
// ===== library types =====

TYPE "LoadDataBlock"
VERSION : 0.1
   STRUCT
      data : Array[0..8192] of USInt;
   END_STRUCT;
END_TYPE

// ===== library: MasterCopy "ReadSDO" =====

FUNCTION_BLOCK "ReadSDO"   // FB104, SCL
{ S7_Optimized_Access := 'TRUE' }
VERSION : 0.1
   VAR_INPUT
      REQ : Bool;   // Start read SDO request
      ID : Word;   // Hardware ID of CM
      SLOT : Byte;   // Channel
      NODE : Int;   // Node ID
      INDEX : Word;   // Object index
      SUB : Byte;   // Object subindex
      DB : DInt;   // First memorybyte where recieved data is stored
   END_VAR
   VAR_OUTPUT
      SIZE : UInt;   // Size of recieved data
      BUSY : Bool;   // FB is busy
      RET : UInt;   // Result
   END_VAR
   VAR
      iState : Int;
      abResponseArray : Array[0..248] of Byte;
      abRequestArray : Array[0..4] of Byte;
      WriteSDO : WRREC;
      ReadSDO : RDREC;
      fReqWriteReadSDO : Bool;
      fReqReadSDO : Bool;
      fWriteReadSDOBusy : Bool;
      fReadSDOBusy : Bool;
      bSubindex : Byte;
      wReturn : Word;
      wErrorCode : Word;
      wNoHammeredSDO : Word;
      iDBIndex : Int;
      uiRequestTotalSize : UInt;
      iResponseDataSize : Int;
      uiResponseTotalSize : UInt;
      bAddErrInfo : Byte;
      dwStatus : DWord;
      fWriteReadSDOError : Bool;
      fWriteReadSDODone : Bool;
      fReadSDOValid : Bool;
      fReadSDOError : Bool;
      uiLen : UInt;
      wLen : Word;
      wTotLen : Word;
      fErrTooMuchSDOData : Bool;
      bNode : Byte;
      wIndex : Word;
      bSub : Byte;
      iReturnSize : Int;
      iDataIndex : Int;
      iResponseHeaderSize : Int;
      iReadLength : Int;
      iRecordNo : Int;
   END_VAR
   VAR_TEMP
      wTemp : Word;
      i : Int;
   END_VAR
BEGIN
   (* ------------------------------------------------------------------------
   Title:        Read SDO
   Description:  Block used for reading a single SDO from any CANopen node.
                 CM CANopen module needs to be in CANopen operation mode. 

   Author:       HMS
   Version:      1.0
   Date:         2013-05-29
      ------------------------------------------------------------------------ *)

   CASE #iState OF
     0:  // START
       IF #REQ THEN
         #BUSY                 :=  true;
         #fReqWriteReadSDO     :=  true;
         #fReqReadSDO          :=  true;

         #fErrTooMuchSDOData    :=  false;

         #fWriteReadSDOBusy    :=  false;
         #fReadSDOBusy         :=  false;

         #bNode                :=  INT_TO_BYTE(#NODE);
         #wIndex               :=  #INDEX;
         #bSub                 :=  #SUB;

         #abRequestArray[0]    :=  0;    //Frag byte
         #iReturnSize          :=  0;
         #iDataIndex           :=  0;

         #uiRequestTotalSize   :=  5;
         #iResponseHeaderSize  :=  9;
         #iResponseDataSize    :=  240;
         #uiResponseTotalSize  :=  249;
         #iRecordNo            :=  WORD_TO_INT(w#16#110);

         #iState               := 10;
     END_IF;

   10: //Check input parameter(s)
       IF #SLOT < 0 OR #SLOT > 7 THEN  // Index should be in the range 0 - 7
         #wReturn      :=  0;
         #bAddErrInfo  :=  B#16#4A;
         #iState       :=  900;  //Internal error
       ELSE
         #iRecordNo    :=  WORD_TO_INT(w#16#110+#SLOT);
         #iState       := 100;  //SDO
       END_IF;      

     100: //SDO
       #wNoHammeredSDO  :=  0;

       // Set up the Read SDO request
       #abRequestArray[1] :=  #bNode;
       #abRequestArray[2] :=  WORD_TO_BYTE(SHR(IN:=#wIndex,N:=8));
       #abRequestArray[3] :=  WORD_TO_BYTE(#wIndex);
       #abRequestArray[4] :=  #bSub;

      #iState   :=  110;

     110:  //Write
       #WriteSDO(
          REQ      :=  #fReqWriteReadSDO,
          ID       :=  #ID,
          INDEX    :=  #iRecordNo,
          LEN      :=  #uiRequestTotalSize,
          DONE     =>  #fWriteReadSDODone,
          BUSY     =>  #fWriteReadSDOBusy,
          ERROR    =>  #fWriteReadSDOError,
          STATUS   =>  #dwStatus,
          RECORD   :=  #abRequestArray
          );

       #fReqWriteReadSDO   :=  false;  // Reset variable to prevent this SFC from being called twice
       IF NOT #fWriteReadSDOBusy THEN
         #iState  := 120;
       END_IF;

     120:  //Evaluate writing
       #wReturn  :=  DWORD_TO_WORD(SHR(IN:=#dwStatus,N:=8)) AND W#16#FFFF;
       IF #fWriteReadSDOError THEN
         #iState  := 903;  //Write error
       ELSE  // Seems no error occured, continue with reading the SDO
         #iState  := 130;   //Read
       END_IF;

     130: //Read
      #ReadSDO(
       REQ       :=  #fReqReadSDO,
       ID        :=  #ID,
       INDEX     :=  #iRecordNo,
       MLEN      :=  #uiResponseTotalSize,
       VALID     =>  #fReadSDOValid,
       BUSY      =>  #fReadSDOBusy,
       ERROR     =>  #fReadSDOError,
       STATUS    =>  #dwStatus,
       LEN       =>  #uiLen,
       RECORD    :=  #abResponseArray
       );

       #fReqReadSDO :=  false;
       IF NOT #fReadSDOBusy THEN
         #iState  := 140;      
       END_IF;

     140:  //Evaluate reading, try again if failed
       #wTemp :=  DWORD_TO_WORD(SHR(IN:=#dwStatus,N:=8)) AND W#16#FFFF;
       IF #wTemp = W#16#80B5 OR #abResponseArray[0] =w#16#FE THEN
         #wNoHammeredSDO  :=  #wNoHammeredSDO + 1;
         IF #wNoHammeredSDO > 1000 THEN
          #wReturn  :=  0;
          #bAddErrInfo :=  b#16#13;
          #iState   := 900;  //Internal error
         ELSE
           #fReqReadSDO    :=  true;
           #iState         := 130;  //Read
         END_IF;
       ELSE
         #iState  := 150;  //CERR
       END_IF;

     150:  //CERR
       IF #fReadSDOError THEN  // Check for failure when sending the command
         #wReturn  :=  DWORD_TO_WORD(SHR(IN:=#dwStatus,N:=8)) AND W#16#FFFF;
         #iState      := 903;  //Read error
        ELSIF #abResponseArray[0] > 0 THEN // Check if the message was rejected by the module
         #wReturn  :=  B#16#FF;
         #bAddErrInfo  :=  #abResponseArray[0];
         #iState      := 903;  //Read error
       ELSE
         #iState  := 160;
     END_IF;

     160:  
       //
       #iReadLength :=  UINT_TO_INT(#uiLen) - #iResponseHeaderSize;
       #iReturnSize :=  #iReturnSize + #iReadLength;

       // Check for SDO error
       IF #abResponseArray[6] <> 0 THEN
         #bAddErrInfo  :=  #abResponseArray[6];
         #wReturn      :=  0;
         #iState       :=  903;
       ELSIF #iDataIndex >= #iResponseDataSize THEN    // Check if the data would be completely outside the array
         #iState       :=  300;  //CONT
       ELSIF (#iDataIndex + #iReadLength) <= #iResponseDataSize THEN
         #iState       :=  200;  //SOK
       ELSE
         #iReadLength  :=  #iResponseDataSize - #iDataIndex;
         #fErrTooMuchSDOData :=  true;
         #iState       :=  200;  //SOK
       END_IF;

     200:  //SOK
       // Copy data to the user-specified array
       FOR #i:=0 TO #iReadLength - 1 DO
         POKE(area       :=  16#84,
              dbNumber   :=  #DB,
              byteOffset :=  #iDataIndex + #i,
              value      :=  #abResponseArray[#iResponseHeaderSize + #i]);
       END_FOR;
       #iDataIndex   :=  #iDataIndex + #iReadLength;
       POKE(area       :=  16#84,
              dbNumber   :=  #DB,
              byteOffset :=  0,
              value      :=  #abResponseArray[#iResponseHeaderSize]);
       #iState       :=  300;  //CONT

     300:  //CONT
       //Check whether OR NOT TO CONTINUE

     // If this was the last message of a fragmented message, or this message was
     //  not fragmented at all, we're done
     IF (#abResponseArray[1] AND 1) = 0 OR (#abResponseArray[1] AND 2) > 0 THEN  
       #iState             := 400;  //DONE
     ELSE    // Not the last fragment, go again!
       #abRequestArray[1]  :=  #abResponseArray[1];
       #fReqWriteReadSDO   :=  true;
       #fReqReadSDO        :=  true;
       #iState             := 100;  //SDO
     END_IF;

     400:  //DONE
       IF #fErrTooMuchSDOData THEN
         #wErrorCode :=  W#16#22;
         #iState     :=  900;
       ELSE
         #RET    :=  0;
         #BUSY   :=  false;
         #SIZE   :=  INT_TO_UINT(#iReturnSize);
         #iState     :=  0;
       END_IF;

   (*** ERROR HANDLING ***)
     900:// Internal errors
       IF #wReturn = 0 AND #bAddErrInfo <> 0 THEN
         #wErrorCode :=  w#16#1000 + #bAddErrInfo;     
       ELSE
         #wErrorCode :=  W#16#FF00;  
       END_IF;
       #iState  := 999;

     903: //Range 3xxx (Read/Write errors)
       IF #wReturn = W#16#8090 THEN
         #wErrorCode :=  W#16#3100;
       ELSIF #wReturn = W#16#8093 THEN
         #wErrorCode :=  W#16#3200;
       ELSIF #wReturn = W#16#80A0 OR #wReturn = W#16#80A1 THEN
         #wErrorCode :=  W#16#3300;
       ELSIF #wReturn = W#16#80A2 THEN
         #wErrorCode :=  W#16#3701;
       ELSIF #wReturn = W#16#80A3 THEN
         #wErrorCode :=  W#16#3600;
       ELSIF #wReturn = W#16#80A4 THEN
         #wErrorCode :=  W#16#3702;
       ELSIF #wReturn = W#16#80B2 THEN
         #wErrorCode :=  W#16#3400;
       ELSIF #wReturn = W#16#80B3 THEN
         #wErrorCode :=  W#16#3500;
       ELSIF #wReturn >= W#16#80C1 AND #wReturn <= W#16#80C6 THEN
         #wErrorCode :=  #wReturn - W#16#80C0 + W#16#3702;
       ELSIF #wReturn = 0 THEN
         #wErrorCode :=  W#16#3800 + #bAddErrInfo;
       ELSIF #wReturn = W#16#FF THEN
         #wErrorCode :=  W#16#3900 + #bAddErrInfo;
       ELSE
         IF #wReturn <> 0 OR #bAddErrInfo = 0 THEN
           #wErrorCode :=  W#16#FF00;
         ELSE
           #wErrorCode :=  SHL(IN:=#bAddErrInfo, N:=8);
         END_IF;
       END_IF;
       #iState :=  999;

     999:
       IF #wErrorCode = 0 THEN
         #RET  :=  WORD_TO_UINT(w#16#FF00);
       ELSE
         #RET  :=  WORD_TO_UINT(#wErrorCode);
       END_IF;
       #SIZE   :=  INT_TO_UINT(#iReturnSize); 
       #BUSY   :=  false;
       #iState := 0;
   END_CASE;
END_FUNCTION_BLOCK

// ===== library: MasterCopy "CAN_CTRL" =====

FUNCTION_BLOCK "CAN_CTRL"   // FB1, SCL
{ S7_Optimized_Access := 'TRUE' }
VERSION : 0.1
   VAR_INPUT
      Req : Bool;
      ID : Word;
      FCN : Int;
      LEN : UInt;
      DB : DInt;
   END_VAR
   VAR_OUTPUT
      Busy : Bool;
      Ret : UInt;
   END_VAR
   VAR
      Read : RDREC;
      Write : WRREC;
      iState : Int;
      fReqWriteCmd : Bool;
      fWriteCmdDone : Bool;
      fWriteCmdBusy : Bool;
      fWriteCmdError : Bool;
      dwStatus : DWord;
      abRequest : Array[0..244] of Byte;
      fReqReadCmd : Bool;
      fReadCmdValid : Bool;
      fReadCmdBusy : Bool;
      fReadCmdError : Bool;
      uiLen : UInt;
      abResponse : Array[0..247] of Byte;
      iResonseHeaderSize : Int := 3;
      iResponseDataSize : Int := 245;
      uiResponseTotalSize : UInt := 248;
      wReturn : Word;
      bAddErrInfo : Byte;
      wNoHammered : Word;
      wErrorCode : Word;
      fHasMoreFragments : Bool;
      wParamLength : Word;
      uiCmdLength : UInt;
      wCOBIDsWritten : Word;
      bFragSegment : Byte;
      iOffset : Int;
      wLength : Word;
      iRecordNo : Int;
   END_VAR
   VAR_TEMP
      wTempStatus : Word;
      wTemp : Word;
      i : Int;
   END_VAR
BEGIN
   (* ------------------------------------------------------------------------
   Title:        CAN Control
   Description:  Block used for controlling a CM CANopen 
                 module in transparent mode

   Author:       HMS
   Version:      1.0
   Date:         2013-05-25
      ------------------------------------------------------------------------ *)

   CASE #iState OF
     0:  // Start a new send, reset variables and go
       IF #Req THEN
         #Busy               :=  true;

         #fReqWriteCmd       :=  true;
         #fWriteCmdDone      :=  false;
         #fWriteCmdBusy      :=  false;
         #fWriteCmdError     :=  false;

         #fHasMoreFragments  :=  false;

         #fReqReadCmd    :=  true;
         #fReadCmdValid  :=  false;
         #fReadCmdBusy   :=  false;
         #fReadCmdError  :=  false;

         #dwStatus       :=  0;
         #wNoHammered    :=  0;
         #uiCmdLength    :=  0;

         #abResponse[0]  :=  0;
         #abResponse[1]  :=  0;
         #abResponse[2]  :=  0;
         #abResponse[3]  :=  0;
         #wCOBIDsWritten :=  0;

         #iRecordNo      :=  WORD_TO_INT(w#16#9A);
         #wLength        :=  UINT_TO_WORD(#LEN);

        // Check that FCN is a valid value (0 - 5) and jump to label for handling
        CASE #FCN OF
           1:  // FCN = 1 - params, go to function 1 handling
             #iState       := 10;
           2:  // FCN = 2 - params, go to function 2 handling
            #iState        := 110;
           3:  //#FCN = 3 - no params, go TO sending the command
             #iState       := 130;
           5:  // FCN = 5 - no params, go to sending the command
             #iState       := 130;
         ELSE
             #wReturn      :=  0;
             #bAddErrInfo  :=  B#16#9B;
             #iState       :=  900;  //Internal error
         END_CASE;       
     END_IF;

     10: //Function 1 - Set acceptance filter
       // Check that LEN is in the valid range 0-2048
       IF #LEN > 0 AND #LEN < 2048 THEN
           #iState       := 40;
       ELSE
         #wReturn      :=  0;
         #bAddErrInfo  :=  B#16#9C;
         #iState       :=  900;  //Internal error
       END_IF;      

     40: // 
       IF #LEN <= 119 THEN        
       // Message fits in one fragment, don't touch the fragmentation byte,
       // since it's already set to 0 (= no fragmentation)
       // Store the number of bytes needed to send the parameters

         #wParamLength   :=  #wLength * 2;

         #fHasMoreFragments  :=  false;

         #iState       :=  100;  //COPY
       ELSE
         #iState       :=  50;   //MORE
       END_IF;      

     50: //MORE
       // More than 119 parameters, then the messages has to be fragmented
       IF #wCOBIDsWritten = 0 THEN
         // Update the fragmentation segment for next fragment
         #bFragSegment  := 1;

         // Store the number of bytes needed to send the parameters
         #wParamLength  :=  238;

         #wCOBIDsWritten     :=  119;
         #fHasMoreFragments  :=  true;

         #iState       :=  100;  //COPY
       ELSE
          #iState       :=  60;   //MID
       END_IF;

     60: //MID
       // Check if this is the last fragment
       IF #wCOBIDsWritten + 119 < #wLength THEN
         // Update the fragmentation segment for next fragment
         #bFragSegment :=  #bFragSegment + 1;

         // Store the number of bytes needed to send the parameters
         #wParamLength  :=  238;

         #wCOBIDsWritten     :=  #wCOBIDsWritten + 119;
         #fHasMoreFragments  :=  true;

         #iState       :=  100;  //COPY
       ELSE
         #iState       :=  70;   //LAST     
       END_IF;

     70: //LAST
      // Update the fragmentation segment for next fragment
       #bFragSegment :=  #bFragSegment + 1;

       // Store the number of bytes needed to send the parameters
       #wParamLength  :=  (#wLength - #wCOBIDsWritten) * 2;

       #fHasMoreFragments  :=  false;

       #iState       :=  100;  //COPY

     100:  //COPY
       #iOffset :=  4; //4 bytes (CAN header = 2 byte, No.of CAN IDs = 2 byte)
       FOR #i := 0 TO WORD_TO_INT(#wParamLength) DO    //Max 238-1 (119) words
         #abRequest[#i+#iOffset]  :=  PEEK(area:=16#84, dbNumber:=#DB, byteOffset:=#i + WORD_TO_INT(#wCOBIDsWritten*2));
       END_FOR;

       // Enter number of COB IDs to the request
       #abRequest[3] :=  WORD_TO_BYTE(#wParamLength / 2);  //No.OF CAN IDs = 2 byte
       #wTemp        :=  #wParamLength / 2;
       #abRequest[2] :=  WORD_TO_BYTE(SHR(IN:=#wTemp, N:=8));

       #iState       :=  150;  //SEND

     110:  //Function 2 - Set buffer limit

       #iOffset :=  2; //2 bytes Header (CAN header = 2 byte)
       FOR #i := 0 TO 1 DO  //Only 1 word
         #abRequest[#i+#iOffset]  :=  PEEK(area:=16#84, dbNumber:=#DB, byteOffset:=#i);
       END_FOR;

       #wParamLength   :=  2;
       #iState         := 150;   //SEND

     130:
       #iOffset        :=  2; //1 bytes Header (CAN header = 1 byte)
       #wParamLength   :=  0;
       #iState         := 150;   //SEND

     150:  //SEND
       //Send control command

       #abRequest[0] :=  INT_TO_BYTE(#FCN);
       #abRequest[1] :=  0;

       #uiCmdLength :=  WORD_TO_UINT(#wParamLength) + INT_TO_UINT(#iOffset);

       #Write(
          REQ      :=  #fReqWriteCmd,
          ID       :=  #ID,
          INDEX    :=  #iRecordNo,
          LEN      :=  #uiCmdLength,
          DONE     =>  #fWriteCmdDone,
          BUSY     =>  #fWriteCmdBusy,
          ERROR    =>  #fWriteCmdError,
          STATUS   =>  #dwStatus,
          RECORD   :=  #abRequest
          );

       #fReqWriteCmd   :=  false;
       IF NOT #fWriteCmdBusy THEN
         #iState  := 155;      
       END_IF;

     155:  //Evaluate writing
       #wReturn  :=  DWORD_TO_WORD(SHR(IN:=#dwStatus,N:=8)) AND W#16#FFFF;
       IF #fWriteCmdError THEN
         #iState  := 903;  //Write error
       ELSE  // Seems no error occured, continue with reading
         #iState  := 160;   //Read
       END_IF;

     160:
       #Read(
         REQ       :=  #fReqReadCmd,
         ID        :=  #ID,
         INDEX     :=  #iRecordNo,
         MLEN      :=  #uiResponseTotalSize,
         VALID     =>  #fReadCmdValid,
         BUSY      =>  #fReadCmdBusy,
         ERROR     =>  #fReadCmdError,
         STATUS    =>  #dwStatus,
         LEN       =>  #uiLen,
         RECORD    :=  #abResponse
         );

       #fReqReadCmd   :=  false;
       IF NOT #fReadCmdBusy THEN
           #iState         := 180;
       END_IF;

     180: //Evaluate reading, try again if failed
      #wTempStatus :=  DWORD_TO_WORD(SHR(IN:=#dwStatus,N:=8)) AND W#16#FFFF;
       IF #wTempStatus = W#16#80B5 OR #abResponse[0] = w#16#FE THEN
         #wNoHammered    :=  #wNoHammered + 1;
         IF #wNoHammered > 1000 THEN
           #wReturn      :=  0;
           #bAddErrInfo  :=  b#16#14;
           #iState       := 900;  //Internal error
         ELSE
           #fReqReadCmd  :=  true;
           #iState       := 155;
         END_IF;
       ELSE
         #iState         := 190;
       END_IF;

     190: // Evaluate reading
         IF #fReadCmdError THEN  // Check for failure when sending the command
           #wReturn      :=  DWORD_TO_WORD(SHR(IN:=#dwStatus,N:=8)) AND W#16#FFFF;
           #iState       := 903;  //Read error
         ELSIF #abResponse[0] > 0 THEN // Check if the message was rejected by the module
           #wReturn  :=  B#16#FF;
           #bAddErrInfo  :=  #abResponse[0];
           #iState       := 903;  //Read error
         ELSIF #fHasMoreFragments THEN //More fragments
           #wReturn      :=  DWORD_TO_WORD(SHR(IN:=#dwStatus,N:=8)) AND W#16#FFFF;
           #iState       := 50;   //MORE
         ELSE // No more fragments - we're done!
           #wReturn      :=  DWORD_TO_WORD(SHR(IN:=#dwStatus,N:=8)) AND W#16#FFFF;        
           #Ret          :=  0;
           #Busy         :=  false;
           #iState       :=  0;  
         END_IF;

   (*** ERROR HANDLING ***)
     900:// Internal errors
       IF #wReturn = 0 AND #bAddErrInfo <> 0 THEN
          #wErrorCode :=  w#16#1000 + #bAddErrInfo;     
      ELSE
         #wErrorCode :=  W#16#FF00;  
       END_IF;
       #iState  := 999;

     903: //Range 3xxx (Read/Write errors)
       IF #wReturn = W#16#8090 THEN
         #wErrorCode :=  W#16#3100;
       ELSIF #wReturn = W#16#8093 THEN
         #wErrorCode :=  W#16#3200;
       ELSIF #wReturn = W#16#80A0 OR #wReturn = W#16#80A1 THEN
         #wErrorCode :=  W#16#3300;
       ELSIF #wReturn = W#16#80A2 THEN
         #wErrorCode :=  W#16#3701;
       ELSIF #wReturn = W#16#80A3 THEN
         #wErrorCode :=  W#16#3600;
       ELSIF #wReturn = W#16#80A4 THEN
         #wErrorCode :=  W#16#3702;
       ELSIF #wReturn = W#16#80B2 THEN
         #wErrorCode :=  W#16#3400;
       ELSIF #wReturn = W#16#80B3 THEN
         #wErrorCode :=  W#16#3500;
       ELSIF #wReturn >= W#16#80C1 AND #wReturn <= W#16#80C6 THEN
         #wErrorCode :=  #wReturn - W#16#80C0 + W#16#3702;
       ELSIF #wReturn = 0 THEN
         #wErrorCode :=  W#16#3800 + #bAddErrInfo;
       ELSIF #wReturn = W#16#FF THEN
         #wErrorCode :=  W#16#3900 + #bAddErrInfo;
       ELSE
         IF #wReturn <> 0 AND #bAddErrInfo = 0 THEN
           #wErrorCode :=  W#16#FF00;
         ELSE
           #wErrorCode :=  SHL(IN:=#bAddErrInfo, N:=8);
         END_IF;
       END_IF;
       #iState :=  999;

     999:
       IF #wErrorCode = 0 THEN
         #Ret  :=  WORD_TO_UINT(w#16#FF00);
       ELSE
         #Ret  :=  WORD_TO_UINT(#wErrorCode);
       END_IF;
       #Busy   :=  false;
       #iState :=  0; 
   END_CASE;
END_FUNCTION_BLOCK

// ===== library: MasterCopy "CAN_RCV" =====

FUNCTION_BLOCK "CAN_RCV"   // FB107, SCL
{ S7_Optimized_Access := 'TRUE' }
VERSION : 0.1
   VAR_INPUT
      REQ : Bool;   // Start recieve
      DB : DInt;   // First memory byte where data in recieved frame is stored
      ID : Word;   // Hardware ID of CM
      ACK : Bool;   // Acknowledge recieved frame
   END_VAR
   VAR_OUTPUT
      BUSY : Bool;   // FB is busy
      RET : UInt;   // Result
      RTR : Bool;   // RTR in recieved frame
      COBID : Word;   // CAN ID in recieved frame
      SIZE : UInt;   // Size of recieved data in frame
      NEW : Bool;   // New frame has arrived
   END_VAR
   VAR
      Read : RDREC;
      wErrorCode : Word;
      wReturn : Word;
      bAddErrInfo : Byte;
      iState : Int;
      fLast : Bool;
      fHasMoreFrames : Bool;
      iCanFrameCount : Int;
      fReqRead : Bool;
      fReadBusy : Bool;
      iRecordNo : Int;
      fReadValid : Bool;
      fReadError : Bool;
      dwStatus : DWord;
      abResponseArray : Array[0..247] of Byte;
      iResponseHeaderSize : Int := 3;
      iResponseMessageSize : Int := 245;
      uiResponseTotalSize : Word := 248;
      uiLen : UInt;
      iNoOfFramesInResponse : Int;
      iOffset : Int;
      iCanFrameByteOffset : Int;
      wNoHammered : Word;
   END_VAR
   VAR_TEMP
      i : Int;
      wTemp : Word;
   END_VAR
BEGIN
   (* ------------------------------------------------------------------------
   Title:        CAN Recieve
   Description:  Block used for receiving transparent CAN messages on a  
                 CM CANopen module in transparent mode

   Author:       HMS
   Version:      1.0
   Date:         2013-05-25
      ------------------------------------------------------------------------ *)

   CASE #iState OF
     0:  // Wait for request of status 
       IF #REQ THEN
         #BUSY           :=  true;
         #wReturn        :=  0;
         #wNoHammered    :=  0;
         #NEW            :=  false;

         #iState         := 100;
       END_IF;

     100: // Read the input data

       // Set up the Send request
        #iRecordNo  :=  WORD_TO_INT(w#16#9B);
        #fReqRead   :=  true;

       #iState            :=  110;

     110:  //Read

       #Read(
       REQ       :=  #fReqRead,
       ID        :=  #ID,
       INDEX     :=  #iRecordNo,
       MLEN      :=  #uiResponseTotalSize,
       VALID     =>  #fReadValid,
       BUSY      =>  #fReadBusy,
       ERROR     =>  #fReadError,
       STATUS    =>  #dwStatus,
       LEN       =>  #uiLen,
       RECORD    :=  #abResponseArray
       );

       #fReqRead :=  false;
       IF NOT #fReadBusy THEN
         #iState  := 140;
       END_IF;

     140:  //Evaluate reading, try again if failed
       #wReturn :=  DWORD_TO_WORD(SHR(IN:=#dwStatus,N:=8)) AND W#16#FFFF;
       IF #wReturn = W#16#80B5 OR #abResponseArray[0] = w#16#FE THEN
         #wNoHammered  :=  #wNoHammered + 1;
         IF #wNoHammered > 1000 THEN
          #wReturn     :=  0;
          #bAddErrInfo :=  b#16#13;
          #iState      := 900;//Internal error
         ELSE
           #fReqRead   :=  true;
           #iState     := 110;  //Read
         END_IF;
       ELSE
         #iState       := 150;  //CERR
       END_IF;

     150:  //CERR
       IF #fReadError THEN  // Check for failure when sending the command
         #wReturn      :=  DWORD_TO_WORD(SHR(IN:=#dwStatus,N:=8)) AND W#16#FFFF;
         #iState       := 903;  //Read error
        ELSIF #abResponseArray[0] > 0 THEN // Check if the message was rejected by the module
         #wReturn      :=  B#16#FF;
         #bAddErrInfo  :=  #abResponseArray[0];
         #iState       := 903;  //Read error
       ELSE
         #iState       := 160;
     END_IF;

     160:  
     //Check number of frames in response
     //1st byte in CAN_RCV response data contains number of frames in buffer
       #iNoOfFramesInResponse  := #abResponseArray[3]; 
       IF #iNoOfFramesInResponse = 0 THEN 
         #BUSY       :=  false;
         #RET        :=  0;
         #iState     :=  0;  //Done   
       ELSIF #iNoOfFramesInResponse > 19 THEN
         #wReturn      :=  0;
         #bAddErrInfo  :=  #abResponseArray[3];
         #iState       :=  903;
       ELSE
         #iResponseHeaderSize    :=  3;
         #iCanFrameCount         :=  0;
         #iCanFrameByteOffset    :=  0;
         #iState                 :=  200;  //COPY
       END_IF;

     200:  //COPY
       // Copy data to the user-specified array. 
       // Byte 1 in CAN_RCV response data contains number of frames in buffer (Byte 5 in total response array)
       // Byte 2-13 in "CAN_Rcv" response #DATA contains first (oldest) frame (Byte 6-17 in total response array)
       // Add 12 bytes to get next frame

       // Byte 2-3 + (x*12) in CAN_RCV response data contains COBID  (Byte 6-7 in total response array)
       #wTemp :=  #abResponseArray[#iResponseHeaderSize + 1 + #iCanFrameByteOffset];
       #wTemp :=  SHL(IN:=#wTemp,N:=8) OR #abResponseArray[#iResponseHeaderSize + 2 + #iCanFrameByteOffset];
       #COBID  :=  #wTemp;

       // Byte 4 in CAN_RCV response data contains RTR  (Byte 8 in total response array)
       #RTR := BYTE_TO_BOOL(#abResponseArray[3 + #iResponseHeaderSize + #iCanFrameByteOffset]);

       // Byte 5 in CAN_RCV response data contains SIZE  (Byte 9 in total response array)
       #SIZE  :=  #abResponseArray[4 + #iResponseHeaderSize + #iCanFrameByteOffset];

       // Byte 6-13 in CAN_RCV response data contains DATA (Byte 10-17 in total response array) 
       IF #SIZE > 0 THEN
         FOR #i:=0 TO UINT_TO_INT(#SIZE)-1 DO
           POKE(area       :=  16#84,
                dbNumber   :=  #DB,
                byteOffset :=  #i,
                value      :=  #abResponseArray[5 + #iResponseHeaderSize + #i + #iCanFrameByteOffset]);
         END_FOR;
       END_IF;

       //Increase frame count and frame offset to get next frame
       #iCanFrameByteOffset  :=  #iCanFrameByteOffset + 12;
       #iCanFrameCount       :=  #iCanFrameCount + 1;
       #NEW                  :=  true;
       #iState               :=  300;  //wait for ack

     300:
       IF #ACK THEN
       //Check if more frames in buffer
         IF #iCanFrameCount >= #iNoOfFramesInResponse THEN
           #BUSY       :=  false;
           #RET        :=  0;
           #NEW        :=  false;
           #iState     :=  0;  //Done
         ELSE
           #NEW        :=  false;
           #iState     :=  200;  //copy next frame
         END_IF;
       END_IF;

   (*** ERROR HANDLING ***)
     900:// Internal errors
       IF #wReturn = 0 AND #bAddErrInfo <> 0 THEN
         #wErrorCode :=  w#16#1000 + #bAddErrInfo;      
       ELSE
         #wErrorCode :=  W#16#FF00;  
       END_IF;
       #iState  := 999;

     903: //Range 3xxx (Read/Write errors)
       IF #wReturn = W#16#8090 THEN
         #wErrorCode :=  W#16#3100;
       ELSIF #wReturn = W#16#8093 THEN
         #wErrorCode :=  W#16#3200;
       ELSIF #wReturn = W#16#80A0 OR #wReturn = W#16#80A1 THEN
         #wErrorCode :=  W#16#3300;
       ELSIF #wReturn = W#16#80A2 THEN
         #wErrorCode :=  W#16#3701;
       ELSIF #wReturn = W#16#80A3 THEN
         #wErrorCode :=  W#16#3600;
       ELSIF #wReturn = W#16#80A4 THEN
         #wErrorCode :=  W#16#3702;
       ELSIF #wReturn = W#16#80B2 THEN
         #wErrorCode :=  W#16#3400;
       ELSIF #wReturn = W#16#80B3 THEN
         #wErrorCode :=  W#16#3500;
       ELSIF #wReturn >= W#16#80C1 AND #wReturn <= W#16#80C6 THEN
         #wErrorCode :=  #wReturn - W#16#80C0 + W#16#3702;
       ELSIF #wReturn = 0 THEN
         #wErrorCode :=  W#16#3800 + #bAddErrInfo;
       ELSIF #wReturn = W#16#FF THEN
         #wErrorCode :=  W#16#3900 + #bAddErrInfo;
       ELSE
         IF #wReturn <> 0 OR #bAddErrInfo = 0 THEN
           #wErrorCode :=  W#16#FF00;
         ELSE
           #wErrorCode :=  SHL(IN:=#bAddErrInfo, N:=8);
         END_IF;
       END_IF;
       #iState :=  999;

     999:
       IF #wErrorCode = 0 THEN
         #RET  :=  WORD_TO_UINT(w#16#FF00);
       ELSE
         #RET  :=  WORD_TO_UINT(#wErrorCode);
       END_IF;
       #BUSY   :=  false;
       #iState := 0;
   END_CASE;
END_FUNCTION_BLOCK

// ===== library: MasterCopy "CAN_SEND" =====

FUNCTION_BLOCK "CAN_SEND"   // FB106, SCL
{ S7_Optimized_Access := 'TRUE' }
VERSION : 0.1
   VAR_INPUT
      REQ : Bool;   // Start send
      RTR : Bool;   // RTR in frame to send
      COBID : Word;   // CAN ID in frame to send
      DB : DInt;   // First Memory byte where to find data to send in frame
      DATASIZE : UInt;   // Size of DATA to send in frame
      ABORT : Bool;   // Abort sending af frames
      ID : Word;   // Hardware ID of CM
   END_VAR
   VAR_OUTPUT
      BUSY : Bool;   // FB is Busy
      RET : UInt;   // Result
   END_VAR
   VAR
      Write : WRREC;
      ReadWrite : RDREC;
      wErrorCode : Word;
      wReturn : Word;
      bAddErrInfo : Byte;
      dOutAddr : DWord;
      abRequestArray : Array[0..228] of Byte;
      iRequestHeaderSize : Int := 0;
      iRequestDataSize : Int := 229;
      uiRequestTotalSize : UInt := 229;
      iState : Int;
      iCanFrameCount : Int;
      fReqWrite : Bool;
      fWriteBusy : Bool;
      fReqReadWrite : Bool;
      fReadWriteBusy : Bool;
      iRecordNo : Int;
      fWriteDone : Bool;
      fWriteError : Bool;
      fReadWriteValid : Bool;
      fReadWriteError : Bool;
      dwStatus : DWord;
      abResponseArray : Array[0..247] of Byte;
      iResponseHeaderSize : Int := 3;
      iResponseDataSize : Int := 245;
      uiResponseTotalSize : UInt := 248;
      wNoHammered : Word;
      uiLen : UInt;
   END_VAR
   VAR_TEMP
      bResult : Byte;
      dwAdress : DWord;
      i : Int;
      fResult_1 : Bool;
      fResult_2 : Bool;
      wResult : Word;
   END_VAR
BEGIN
   (* ------------------------------------------------------------------------
   Title:        CAN Send
   Description:  Block FOR sending transparent CAN messages on a 
                 CM CANopen module in transparent mode

   Author:       HMS
   Version:      1.0
   Date:         2013-05-25
      ------------------------------------------------------------------------ *)

   CASE #iState OF
     0:  // Wait for request of status 
       IF #REQ THEN
         #BUSY           :=  true;
         #fReqWrite      :=  true;
         #fReqReadWrite  :=  true;

         #fWriteBusy     :=  false;
         #fReadWriteBusy :=  false;

         #wReturn         :=  0;

         #iState          := 10;  
       END_IF;

     10: // Check whether the COB ID valid
     IF #COBID >= 0 AND #COBID <= W#16#7FF THEN
       #iState       := 40;
     ELSE
       #wReturn      :=  0;
       #bAddErrInfo  :=  B#16#98;
       #iState       :=  900;
     END_IF;

     // Check CAN FRAME Count
       #iCanFrameCount :=  1;

     40: // Check whether the size of the data is valid
     IF #DATASIZE >= 0 AND #DATASIZE <=8 THEN
       #iState       := 100;
     ELSE
       #wReturn      :=  0;
       #bAddErrInfo  :=  B#16#9A;
       #iState       :=  900;
     END_IF;

     100: //

       // Set up the Send request
       #iRecordNo  :=  WORD_TO_INT(w#16#9C);

       //CAN data header
       #abRequestArray[0] :=  INT_TO_BYTE(#iCanFrameCount);
       #abRequestArray[1] :=  WORD_TO_BYTE(SHR(IN:=#COBID,N:=8));
       #abRequestArray[2] :=  WORD_TO_BYTE(#COBID);
       #abRequestArray[3] :=  BOOL_TO_BYTE(#RTR);
       #abRequestArray[4] :=  UINT_TO_BYTE(#DATASIZE);

       //CAN_SND request data (byte 6-13)
       FOR #i:=0 TO UINT_TO_INT(#DATASIZE) - 1 DO
         #abRequestArray[#iCanFrameCount + #iRequestHeaderSize + 4 + #i] := PEEK(
                                                             area       :=  16#84, 
                                                             dbNumber   :=  #DB,
                                                             byteOffset :=  #i
                                                             );
       END_FOR;

       #uiRequestTotalSize  :=  INT_TO_UINT(#iCanFrameCount + #iRequestHeaderSize + 4 + 8);
       #wNoHammered :=  0;

       #iState   :=  110;

     110:  //Write

       #Write(
          REQ      :=  #fReqWrite,
          ID       :=  #ID,
          INDEX    :=  #iRecordNo,
          LEN      :=  #uiRequestTotalSize,
          DONE     =>  #fWriteDone,
          BUSY     =>  #fWriteBusy,
          ERROR    =>  #fWriteError,
          STATUS   =>  #dwStatus,
          RECORD   :=  #abRequestArray
          );

       #fReqWrite   :=  false;  // Reset variable to prevent this SFC from being called twice
       IF NOT #fWriteBusy THEN
         #iState  := 120;
       END_IF;

     120:  //Evaluate writing
       #wReturn  :=  DWORD_TO_WORD(SHR(IN:=#dwStatus,N:=8)) AND W#16#FFFF;
       IF #fWriteError THEN
         #iState  := 903;  //Write error
       ELSE  // Seems no error occured, continue with reading
        #iState  := 130;   //Read
       END_IF;

     130: //Read

       #ReadWrite(
       REQ       :=  #fReqReadWrite,
       ID        :=  #ID,
       INDEX     :=  #iRecordNo,
       MLEN      :=  #uiResponseTotalSize,
       VALID     =>  #fReadWriteValid,
       BUSY      =>  #fReadWriteBusy,
       ERROR     =>  #fReadWriteError,
       STATUS    =>  #dwStatus,
       LEN       =>  #uiLen,
       RECORD    :=  #abResponseArray
       );

       #fReqReadWrite :=  false;
       IF NOT #fReadWriteBusy THEN
         #iState  := 140;      
       END_IF;

     140:  //Evaluate reading, try again if failed
       #wReturn :=  DWORD_TO_WORD(SHR(IN:=#dwStatus,N:=8)) AND W#16#FFFF;
       IF #wReturn = W#16#80B5 OR #abResponseArray[0] = w#16#FE THEN
         #wNoHammered  :=  #wNoHammered + 1;
         IF #wNoHammered > 1000 THEN
          #wReturn     :=  0;
          #bAddErrInfo :=  b#16#13;
          #iState      := 900;  //Internal error
         ELSE
           #fReqReadWrite  :=  true;
           #iState         := 130;  //Read
         END_IF;
       ELSE
         #iState  := 150;  //CERR
       END_IF;

     150:  //CERR
       IF #fReadWriteError THEN  // Check for failure when sending the command
         #wReturn  :=  DWORD_TO_WORD(SHR(IN:=#dwStatus,N:=8)) AND W#16#FFFF;
         #iState      := 903;  //Read error
        ELSIF #abResponseArray[0] > 0 THEN // Check if the message was rejected by the module
         #wReturn      :=  B#16#FF;
         #bAddErrInfo  :=  #abResponseArray[0];
         #iState       := 903;  //Read error
       ELSE
         #RET    :=  0;
         #BUSY   :=  false;
        #iState  := 0;
     END_IF;

     (*** ERROR HANDLING ***)
     900:// Internal errors
       IF #wReturn = 0 AND #bAddErrInfo <> 0 THEN
         #wErrorCode :=  w#16#1000 + #bAddErrInfo;     
       ELSE
         #wErrorCode :=  W#16#FF00;  
       END_IF;
       #iState  := 999;

     903: //Range 3xxx (Read/Write errors)
       IF #wReturn = W#16#8090 THEN
         #wErrorCode :=  W#16#3100;
       ELSIF #wReturn = W#16#8093 THEN
         #wErrorCode :=  W#16#3200;
       ELSIF #wReturn = W#16#80A0 OR #wReturn = W#16#80A1 THEN
         #wErrorCode :=  W#16#3300;
       ELSIF #wReturn = W#16#80A2 THEN
         #wErrorCode :=  W#16#3701;
       ELSIF #wReturn = W#16#80A3 THEN
         #wErrorCode :=  W#16#3600;
       ELSIF #wReturn = W#16#80A4 THEN
         #wErrorCode :=  W#16#3702;
       ELSIF #wReturn = W#16#80B2 THEN
         #wErrorCode :=  W#16#3400;
       ELSIF #wReturn = W#16#80B3 THEN
         #wErrorCode :=  W#16#3500;
       ELSIF #wReturn >= W#16#80C1 AND #wReturn <= W#16#80C6 THEN
         #wErrorCode :=  #wReturn - W#16#80C0 + W#16#3702;
       ELSIF #wReturn = 0 THEN
         #wErrorCode :=  W#16#3800 + #bAddErrInfo;
       ELSIF #wReturn = W#16#FF THEN
         #wErrorCode :=  W#16#3900 + #bAddErrInfo;
       ELSE
         IF #wReturn <> 0 OR #bAddErrInfo = 0 THEN
           #wErrorCode :=  W#16#FF00;
         ELSE
           #wErrorCode :=  SHL(IN:=#bAddErrInfo, N:=8);
         END_IF;
       END_IF;
       #iState :=  999;

     999:
       IF #wErrorCode = 0 THEN
         #RET  :=  WORD_TO_UINT(w#16#FF00);
       ELSE
         #RET  :=  WORD_TO_UINT(#wErrorCode);
       END_IF;
       #BUSY   :=  false;
       #iState := 0;
   END_CASE;
END_FUNCTION_BLOCK

// ===== library: MasterCopy "WriteSDO" =====

FUNCTION_BLOCK "WriteSDO"   // FB105, SCL
{ S7_Optimized_Access := 'TRUE' }
VERSION : 0.1
   VAR_INPUT
      REQ : Bool;   // Start write SDO request
      ID : Word;   // Hardware ID of CM
      SLOT : Byte;   // Channel
      NODE : Int;   // Node ID
      INDEX : Word;   // Object index
      SUB : Byte;   // Object subindex
      DB : DInt;   // First memory byte where to find data to send
      DATASIZE : UInt;   // Size of DATA to send
   END_VAR
   VAR_OUTPUT
      BUSY : Bool;   // FB is busy
      RET : UInt;   // Result
   END_VAR
   VAR
      iState : Int;
      abRequestArray : Array[0..238] of Byte;
      abWriteSDOResp : Array[0..8] of Byte;
      WriteSDO : WRREC;
      ReadSDO : RDREC;
      fReqReadWriteSDO : Bool;
      fReqWriteSDO : Bool;
      fReadWriteSDOBusy : Bool;
      fWriteSDOBusy : Bool;
      bSubindex : Byte;
      wReturn : Word;
      wErrorCode : Word;
      wNoHammeredSDO : Word;
      iDBIndex : Int;
      uiResponseTotalSize : UInt;
      uiSDOMaxSize : UInt;
      bAddErrInfo : Byte;
      dwStatus : DWord;
      fWriteSDOError : Bool;
      fWriteSDODone : Bool;
      fReadWriteSDOValid : Bool;
      fReadWriteSDOError : Bool;
      uiLen : UInt;
      wLen : Word;
      wTotLen : Word;
      bNode : Byte;
      wIndex : Word;
      bSub : Byte;
      wReturnSize : Word;
      iDataIndex : Int;
      uiRequestHeaderSize : UInt;
      uiRequestDataSize : UInt;
      uiRequestTotalSize : UInt;
      iRecordNo : Int;
   END_VAR
   VAR_TEMP
      wTemp : Word;
      i : Int;
   END_VAR
BEGIN
   (* ------------------------------------------------------------------------
   Title:        Write SDO
   Description:  Block used for writing a single SDO to any CANopen node.
                 CM CANopen module needs to be in CANopen operation mode. 

   Author:       HMS
   Version:      1.0
   Date:         2013-05-29
      ------------------------------------------------------------------------ *)

   CASE #iState OF
     0:  // START
       IF #REQ THEN
         #BUSY                 :=  true;
         #fReqReadWriteSDO     :=  true;
         #fReqWriteSDO         :=  true;
         #fReadWriteSDOBusy    :=  false;
         #fWriteSDOBusy        :=  false;

         #bNode                :=  INT_TO_BYTE(#NODE);
         #wIndex               :=  #INDEX;
         #bSub                 :=  #SUB;
         #iDataIndex           :=  0;

         #uiResponseTotalSize  :=  9;
         #uiSDOMaxSize          :=  232;
         #uiRequestHeaderSize   :=  7;
         #iRecordNo            :=  WORD_TO_INT(w#16#100);

         #iState               := 10;
     END_IF;

   10: //Check input parameter(s)
       IF #SLOT < 0 OR #SLOT > 7 THEN  // Slot should be in the range 0 - 7
         #wReturn      :=  0;
         #bAddErrInfo  :=  B#16#4A;
         #iState       :=  900;  //Internal error
       ELSE
         #iRecordNo  :=  WORD_TO_INT(w#16#100 + #SLOT);
         #iState       := 20;  //SDO
       END_IF;      

     20: //WSDO
       #wNoHammeredSDO :=  0;
       IF #DATASIZE > #uiSDOMaxSize THEN
         #iState             := 30; //MORE
       ELSE  
         #uiRequestDataSize       :=  #DATASIZE;
         #abRequestArray[0]  :=  0;
         #iState             := 100;  //SDO
       END_IF;

     30: //MORE
       IF #iDataIndex <> 0  THEN
         #iState             := 40; //BFRE
       ELSE
         #abRequestArray[0]  :=  B#16#15;
         #uiRequestDataSize       :=  #uiSDOMaxSize;
         #iState             :=  100;  //SDO
       END_IF;

     40: //BFRE
       IF (#DATASIZE - INT_TO_UINT(#iDataIndex)) <= #uiSDOMaxSize THEN  //LAST
         #abRequestArray[0]  :=  ((#abRequestArray[0] AND B#16#FB) + b#16#10) OR B#16#2;
         #uiRequestDataSize   :=  #DATASIZE - INT_TO_UINT(#iDataIndex);
         #iState           :=  100;   //SDO
       ELSE
         #abRequestArray[0]  :=  (#abRequestArray[0] AND B#16#FB) + b#16#10;
         #uiRequestDataSize   :=  #uiSDOMaxSize;
         #iState             :=  100;  //SDO
       END_IF;

     100: //SDO

      // Set up the Write SDO request
       #abRequestArray[1] :=  #bNode;
       #abRequestArray[2] :=  WORD_TO_BYTE(SHR(IN:=#wIndex,N:=8));
       #abRequestArray[3] :=  WORD_TO_BYTE(#wIndex);
       #abRequestArray[4] :=  #bSub;
       #abRequestArray[5] :=  WORD_TO_BYTE(SHR(IN:=UINT_TO_WORD(#DATASIZE),N:=8));
       #abRequestArray[6] :=  UINT_TO_BYTE(#DATASIZE);

       FOR #i:=0 TO UINT_TO_INT(#uiRequestDataSize) - 1 DO
         #abRequestArray[UINT_TO_INT(#uiRequestHeaderSize) + #i] := PEEK(area       :=  16#84, 
                                                        dbNumber   :=  #DB,
                                                        byteOffset :=  #iDataIndex + #i
                                                         );
       END_FOR;

       #uiRequestTotalSize  :=  #uiRequestDataSize + #uiRequestHeaderSize;

       #iState   :=  110;

     110:  //Write
       #WriteSDO(
          REQ      :=  #fReqWriteSDO,
          ID       :=  #ID,
          INDEX    :=  #iRecordNo,
          LEN      :=  #uiRequestTotalSize,
          DONE     =>  #fWriteSDODone,
          BUSY     =>  #fWriteSDOBusy,
          ERROR    =>  #fWriteSDOError,
          STATUS   =>  #dwStatus,
          RECORD   :=  #abRequestArray
          );

       #fReqWriteSDO   :=  false;  // Reset variable to prevent this SFC from being called twice
       IF NOT #fWriteSDOBusy THEN
         #iState  := 120;
       END_IF;

     120:  //Evaluate writing
       #wReturn  :=  DWORD_TO_WORD(SHR(IN:=#dwStatus,N:=8)) AND W#16#FFFF;
       IF #fWriteSDOError THEN
         #iState  := 903;  //Write error
       ELSE  // Seems no error occured, continue with reading the SDO
         #iState  := 130;   //Read
       END_IF;

     130: //Read
       #ReadSDO(
         REQ       :=  #fReqReadWriteSDO,
         ID        :=  #ID,
         INDEX     :=  #iRecordNo,
         MLEN      :=  #uiResponseTotalSize,
         VALID     =>  #fReadWriteSDOValid,
         BUSY      =>  #fReadWriteSDOBusy,
         ERROR     =>  #fReadWriteSDOError,
         STATUS    =>  #dwStatus,
         LEN       =>  #uiLen,
         RECORD    :=  #abWriteSDOResp
         );

       #fReqReadWriteSDO :=  false;
       IF NOT #fReadWriteSDOBusy THEN
         #iState  := 140;      
       END_IF;

     140:  //Evaluate reading, try again if failed
       #wTemp :=  DWORD_TO_WORD(SHR(IN:=#dwStatus,N:=8)) AND W#16#FFFF;
       IF #wTemp = W#16#80B5 OR #abWriteSDOResp[0] = w#16#FE THEN
         #wNoHammeredSDO  :=  #wNoHammeredSDO + 1;
         IF #wNoHammeredSDO > 1000 THEN
          #wReturn  :=  0;
          #bAddErrInfo :=  b#16#13;
          #iState   := 900;  //Internal error
         ELSE
           #fReqReadWriteSDO    :=  true;
           #iState         := 130;  //Read
         END_IF;
       ELSE
         #iState  := 150;  //CERR
       END_IF;

     150:  //CERR
       IF #fReadWriteSDOError THEN  // Check for failure when sending the command
         #wReturn  :=  DWORD_TO_WORD(SHR(IN:=#dwStatus,N:=8)) AND W#16#FFFF;
         #iState      := 903;  //Read error
        ELSIF #abWriteSDOResp[0] > 0 THEN // Check if the message was rejected by the module
         #wReturn  :=  B#16#FF;
         #bAddErrInfo  :=  #abWriteSDOResp[0];
         #iState      := 903;  //Read error
       ELSE
         #iState  := 160;
     END_IF;

     160:  
       // Check for SDO error
       IF #abWriteSDOResp[6] <> 0 THEN
         #bAddErrInfo  :=  #abWriteSDOResp[6];
         #wReturn      :=  0;
         #iState       :=  903;
       ELSE
         #iDataIndex  :=  #iDataIndex + UINT_TO_INT(#uiRequestDataSize);
         #iState       :=  300;  //CONT
       END_IF;

     300:  //CONT
       //Check whether OR NOT TO CONTINUE

     // If this was the last message of a fragmented message, or this message was
     //  not fragmented at all, we're done
     IF (#abRequestArray[0] AND 1) = 0 OR (#abRequestArray[0] AND 2) > 0 THEN
       #iState  := 400;  //DONE
     ELSE    // Not the last fragment, go again!
       #fReqWriteSDO      :=  true;
       #fReqReadWriteSDO :=  true;
       #iState  := 100;  //SDO
     END_IF;

     400:  //DONE
       #RET    :=  0;
       #BUSY   :=  false;
       #iState  := 0;

   (*** ERROR HANDLING ***)
     900:// Internal errors
       IF #wReturn = 0 AND #bAddErrInfo <> 0 THEN
         #wErrorCode :=  w#16#1000 +#bAddErrInfo;     
       ELSE
         #wErrorCode :=  W#16#FF00;  
       END_IF;
       #iState  := 999;

     903: //Range 3xxx (Read/Write errors)
       IF #wReturn = W#16#8090 THEN
         #wErrorCode :=  W#16#3100;
       ELSIF #wReturn = W#16#8093 THEN
         #wErrorCode :=  W#16#3200;
       ELSIF #wReturn = W#16#80A0 OR #wReturn = W#16#80A1 THEN
         #wErrorCode :=  W#16#3300;
       ELSIF #wReturn = W#16#80A2 THEN
         #wErrorCode :=  W#16#3701;
       ELSIF #wReturn = W#16#80A3 THEN
         #wErrorCode :=  W#16#3600;
       ELSIF #wReturn = W#16#80A4 THEN
         #wErrorCode :=  W#16#3702;
       ELSIF #wReturn = W#16#80B2 THEN
         #wErrorCode :=  W#16#3400;
       ELSIF #wReturn = W#16#80B3 THEN
         #wErrorCode :=  W#16#3500;
       ELSIF #wReturn >= W#16#80C1 AND #wReturn <= W#16#80C6 THEN
         #wErrorCode :=  #wReturn - W#16#80C0 + W#16#3702;
       ELSIF #wReturn = 0 THEN
         #wErrorCode :=  W#16#3800 + #bAddErrInfo;
       ELSIF #wReturn = W#16#FF THEN
         #wErrorCode :=  W#16#3900 + #bAddErrInfo;
       ELSE
         IF #wReturn <> 0 OR #bAddErrInfo = 0 THEN
           #wErrorCode :=  W#16#FF00;
         ELSE
           #wErrorCode :=  SHL(IN:=#bAddErrInfo, N:=8);
         END_IF;
       END_IF;
       #iState :=  999;

     999:
     IF #wErrorCode = 0 THEN
       #RET  :=  WORD_TO_UINT(w#16#FF00);
     ELSE
       #RET  :=  WORD_TO_UINT(#wErrorCode);
     END_IF;
       #BUSY :=  false;
       #iState := 0;
   END_CASE;
END_FUNCTION_BLOCK